FUNCTION_BLOCK FB_Generator_Square
VAR_INPUT
END_VAR
VAR_OUTPUT
END_VAR
VAR
END_VAR

END_FUNCTION_BLOCK

(* stored: Version 1.1.0.1, ProductVersion 3.1.4024.13
   POU FB_Generator_Square: Id {56bac490-8773-4d84-b773-ccc156e890f2}, SpecialFunc None *)
